// TIA Portal project "Beleuchtungsanlage_v1" (V20)

(* hardware
DEVICE "S7-1500/ET200MP-Station_1"  S7-1500 station
   slot 0: "Profilschiene_0"  Rack  6ES7 590-1***0-0AA0
   slot 1: "PLC_1"  CPU 1513-1 PN  6ES7 513-1AM03-0AB0  V4.0
      slot 3: "CPU-Display_1"  6ES7591-1AA00-0AA0
      slot 32768: "PROFINET-Schnittstelle_1"  X1
         slot 32769: "Port_1"  X1 P1
         slot 32770: "Port_2"  X1 P2
      slot 34817: "Virtual CP interface port_1"  Virtual CP interface port  Virtual CP interface port FW V4.0
   slot 2: "DI 16x24VDC BA_1"  DI 16x24VDC BA  6ES7 521-1BH10-0AA0  V1.1
   slot 3: "DQ 16x24VDC/0.5A ST_1"  DQ 16x24VDC/0.5A ST  6ES7 522-1BH00-0AB0  V2.0
   slot 4: "AI 8xU/I/R/RTD BA_1"  AI 8xU/I/R/RTD BA  6ES7 531-7QF00-0AB0  V1.0
   slot 5: "AQ 8xU/I HS_1"  AQ 8xU/I HS  6ES7 532-5HF00-0AB0  V2.2
*)

// ===== PLC "PLC_1"  CPU 1513-1 PN =====

VAR_GLOBAL   // PLC tag table "Standard-Variablentabelle"
   "PlcLabConnectIn01" AT %ID32760 : DWord;
   "PlcLabConnectIn02" AT %ID32764 : DWord;
   "PlcLabConnectOut01" AT %QD32760 : DWord;
   "PlcLabConnectOut02" AT %QD32764 : DWord;
   "Grundstellung" AT %M1.0 : Bool;
   "Zaehler" AT %MW2 : Int;
   "Hochzaehlen" AT %M1.1 : Bool;
   "Runterzaehlen" AT %M1.2 : Bool;
   "Seq_hoch" AT %M1.3 : Bool;
   "Seq_runter" AT %M1.4 : Bool;
   "Tag_2" AT %M3.0 : Bool;
   "Tag_3" AT %M3.1 : Bool;
   "Drei_erreicht" AT %M3.2 : Bool;
   "Null_erreicht" AT %M3.3 : Bool;
END_VAR

VAR_GLOBAL   // PLC tag table "Eingaenge"
   "S2" AT %E0.0 : Bool;
   "Anlage_ein" AT %E0.1 : Bool;
END_VAR

VAR_GLOBAL   // PLC tag table "Ausgaenge"
   "H1" AT %A0.0 : Bool;
   "H2" AT %A0.1 : Bool;
   "H3" AT %A0.2 : Bool;
END_VAR

// folder: System blocks/Program resources

DATA_BLOCK "IEC_Counter_0_DB"   // DB1
{ S7_Optimized_Access := 'TRUE' }
AUTHOR : Simatic
FAMILY : IEC
NAME : CNTR
VERSION : 1.0
// stored: InstanceOfName IEC_COUNTER
"IEC_COUNTER"
BEGIN
END_DATA_BLOCK

// folder: (top level)

FUNCTION "Beleuchtungsanlage" : Void   // FC1, FBD
{ S7_Optimized_Access := 'TRUE' }
VERSION : 0.1
BEGIN

REGION Network 1: Zustände
   // Wenn Zustand eins (1, 5) aktiv ist, dann soll nur Lampe H1 leuchten.
   // Wenn Zustand zwei (2, 4) aktiv ist, dann soll Lampe H1 und H2 leuchten.
   // Wenn Zustand drei (3) aktiv ist, dann sollen alle Lampen (H1, H2 und H3) leuchten.
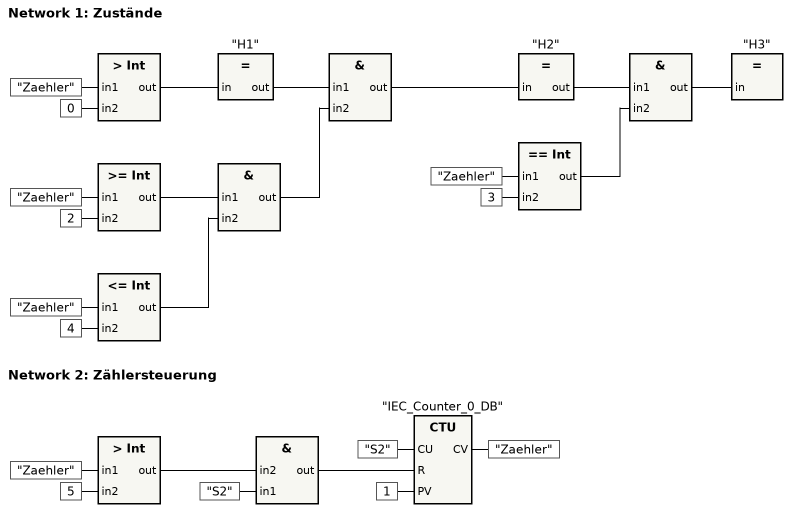
   "H1" := "Zaehler" > 0;
   "H2" := "H1" AND ("Zaehler" >= 2) AND ("Zaehler" <= 4);
   "H3" := "H2" AND ("Zaehler" = 3);
END_REGION

REGION Network 2: Zählersteuerung
   // Beim drücken des Tasters, zählt der Zähler bis zur 5 hoch. Danach wird der Zähler (beim 6.-mal drücken) zurückgesetzt.
   "IEC_Counter_0_DB".CTU(CU := "S2", R := ("Zaehler" > 5) AND "S2", PV := 1, CV => "Zaehler");
END_REGION
END_FUNCTION

ORGANIZATION_BLOCK "Main"   // OB1, FBD, ProgramCycle
TITLE = "Main Program Sweep (Cycle)"
{ S7_Optimized_Access := 'TRUE' }
VERSION : 0.1
   VAR_INPUT
      Initial_Call : Bool;   // Initial call of this OB
      Remanence : Bool;   // =True, if remanent data are available
   END_VAR
BEGIN

REGION Network 1
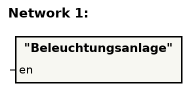
   "Beleuchtungsanlage"();
END_REGION
END_ORGANIZATION_BLOCK